# EPICS StreamDevice protocol: support/stream/StreamDevice/streamApp/simple.proto
terminator = CR LF;

cmd {
    out "%s";
}
info {
    extrainput=ignore;
    out "%s";
    in "%39c";
}
read {
    in "%39c";
}
